(* PLC project Generated.project, CODESYS CODESYS V3.5 SP19 Patch 1 *)
(* stored: creationDateTime 2026-09-01T00:57:57.811073, modificationDateTime 2026-09-01T00:57:57.811073 *)

(* ═══════════════════════════════════════════════════════════════ 🪨 ST_CycleExtractionHMI — Échange IHM cycle extraction ═══════════════════════════════════════════════════════════════ *)
TYPE ST_CycleExtractionHMI : STRUCT
  Cmd : ST_CycleExtractionCmd;
  State : ST_CycleExtractionState;
  Cfg : ST_CycleExtractionCfg;
END_STRUCT;
END_TYPE

(* ═══════════════════════════════════════════════════════════════ ⚙️ ST_CycleExtractionCfg — Réglages persistants cycle extraction 📄 Doc : DOC/AF/AF_Partie-04_Mode_SemiAuto_Sequenceur_v2.3.md §3ter ═══════════════════════════════════════════════════════════════ *)
TYPE ST_CycleExtractionCfg : STRUCT
  ExtractionControlDistance_M : REAL := 2;  (* Remontée palier 1 avant accélération *)
  Initialized : BOOL := FALSE;  (* 🚦 flag restauration boot *)
END_STRUCT;
END_TYPE

(* ═══════════════════════════════════════════════════════════════ 🎮 ST_CycleExtractionCmd — Sélections IHM cycle extraction ═══════════════════════════════════════════════════════════════ *)
TYPE ST_CycleExtractionCmd : STRUCT
  TglEnableExtractionSequence : BOOL := FALSE;  (* Assistance extraction active *)
END_STRUCT;
END_TYPE

(* ═══════════════════════════════════════════════════════════════ 🚦 ST_CycleExtractionState — États publics cycle extraction ═══════════════════════════════════════════════════════════════ *)
TYPE ST_CycleExtractionState : STRUCT
  ExtractionReady : BOOL;
  ExtractionBusy : BOOL;
  ExtractionDone : BOOL;
  ExtractionError : BOOL;
  ExtractionErrorId : WORD;
  ExtractionState : E_ExtractionAssistState;
  ExtractionStepAtFault : E_ExtractionAssistState;
END_STRUCT;
END_TYPE
